FUNCTION_BLOCK Calculator
  (* Standard: 61499-2 *)
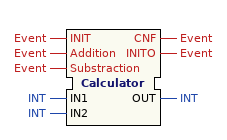
  EVENT_INPUT
    INIT;
    Addition;
    Substraction;
  END_EVENT
  EVENT_OUTPUT
    CNF;
    INITO;
  END_EVENT
  VAR_INPUT
    IN1 : INT;
    IN2 : INT;
  END_VAR
  VAR_OUTPUT
    OUT : INT;
  END_VAR
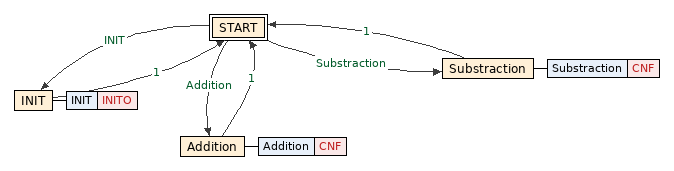
  EC_STATES
    START;
    INIT : INIT -> INITO;
    Addition : Addition -> CNF;
    Substraction : Substraction -> CNF;
  END_STATES
  EC_TRANSITIONS
    START TO INIT := INIT;
    INIT TO START := 1;
    START TO Addition := Addition;
    Addition TO START := 1;
    START TO Substraction := Substraction;
    Substraction TO START := 1;
  END_TRANSITIONS
  ALGORITHM INIT IN ST:
OUT := 0;&#10;
  END_ALGORITHM
  ALGORITHM Addition IN ST:
OUT := IN1 + IN2;&#10;
  END_ALGORITHM
  ALGORITHM Substraction IN ST:
OUT := IN1 - IN2;&#10;
  END_ALGORITHM
END_FUNCTION_BLOCK
